TYPE ST_HmiComm :
STRUCT
	udiHeartbeat : UDINT;   // HMI周期递增
    bOnline      : BOOL;    // PLC判断HMI是否在线
    bTimeout     : BOOL;    // PLC判断通信是否超时
END_STRUCT
END_TYPE

(* stored: Version 1.1.0.1, ProductVersion 3.1.4026.18
   DUT ST_HmiComm: Id {7cbae786-3eef-4a6a-889b-2a0e2ec633b0} *)
